TYPE MDP5001_342_I_066CA8C6 :
STRUCT
	MDP5001_342_I1_Channel_Overcurrent						: BIT;
	MDP5001_342_I1_Channel_Inaccurate_Current				: BIT;
	MDP5001_342_I1_Channel_Current_Guard_Warning			: BIT;
	MDP5001_342_I1_Channel_Current_Guard_Error				: BIT;
	MDP5001_342_I1_Channel_Apparent_Power_Guard_Warning		: BIT;
	MDP5001_342_I1_Channel_Apparent_Power_Guard_Error		: BIT;
	MDP5001_342_I1_Channel_Active_Power_Guard_Warning		: BIT;
	MDP5001_342_I1_Channel_Active_Power_Guard_Error			: BIT;
	MDP5001_342_I1_Channel_Reactive_Power_Guard_Warning		: BIT;
	MDP5001_342_I1_Channel_Reactive_Power_Guard_Error		: BIT;
	MDP5001_342_I1_Channel_DPM_Inaccurate					: BIT;
	MDP5001_342_I1_Channel_DPM_Timeout						: BIT;
	MDP5001_342_I1_Channel_TxPDO_Toggle						: BIT;
	MDP5001_342_I1_Channel_Current							: REAL;
	MDP5001_342_I1_Channel_Active_Power						: REAL;
	MDP5001_342_I1_Channel_Apparent_Power					: REAL;
	MDP5001_342_I1_Channel_Reactive_Power_Fundamental		: REAL;
	MDP5001_342_I1_Channel_Active_Energy					: DINT;
	MDP5001_342_I2_Channel_Overcurrent						: BIT;
	MDP5001_342_I2_Channel_Inaccurate_Current				: BIT;
	MDP5001_342_I2_Channel_Current_Guard_Warning			: BIT;
	MDP5001_342_I2_Channel_Current_Guard_Error				: BIT;
	MDP5001_342_I2_Channel_Apparent_Power_Guard_Warning		: BIT;
	MDP5001_342_I2_Channel_Apparent_Power_Guard_Error		: BIT;
	MDP5001_342_I2_Channel_Active_Power_Guard_Warning		: BIT;
	MDP5001_342_I2_Channel_Active_Power_Guard_Error			: BIT;
	MDP5001_342_I2_Channel_Reactive_Power_Guard_Warning		: BIT;
	MDP5001_342_I2_Channel_Reactive_Power_Guard_Error		: BIT;
	MDP5001_342_I2_Channel_DPM_Inaccurate					: BIT;
	MDP5001_342_I2_Channel_DPM_Timeout						: BIT;
	MDP5001_342_I2_Channel_TxPDO_Toggle						: BIT;
	MDP5001_342_I2_Channel_Current							: REAL;
	MDP5001_342_I2_Channel_Active_Power						: REAL;
	MDP5001_342_I2_Channel_Apparent_Power					: REAL;
	MDP5001_342_I2_Channel_Reactive_Power_Fundamental		: REAL;
	MDP5001_342_I2_Channel_Active_Energy					: DINT;
	MDP5001_342_I3_Channel_Overcurrent						: BIT;
	MDP5001_342_I3_Channel_Inaccurate_Current				: BIT;
	MDP5001_342_I3_Channel_Current_Guard_Warning			: BIT;
	MDP5001_342_I3_Channel_Current_Guard_Error				: BIT;
	MDP5001_342_I3_Channel_Apparent_Power_Guard_Warning		: BIT;
	MDP5001_342_I3_Channel_Apparent_Power_Guard_Error		: BIT;
	MDP5001_342_I3_Channel_Active_Power_Guard_Warning		: BIT;
	MDP5001_342_I3_Channel_Active_Power_Guard_Error			: BIT;
	MDP5001_342_I3_Channel_Reactive_Power_Guard_Warning		: BIT;
	MDP5001_342_I3_Channel_Reactive_Power_Guard_Error		: BIT;
	MDP5001_342_I3_Channel_DPM_Inaccurate					: BIT;
	MDP5001_342_I3_Channel_DPM_Timeout						: BIT;
	MDP5001_342_I3_Channel_TxPDO_Toggle						: BIT;
	MDP5001_342_I3_Channel_Current							: REAL;
	MDP5001_342_I3_Channel_Active_Power						: REAL;
	MDP5001_342_I3_Channel_Apparent_Power					: REAL;
	MDP5001_342_I3_Channel_Reactive_Power_Fundamental		: REAL;
	MDP5001_342_I3_Channel_Active_Energy					: DINT;	
	MDP5001_342_I4_Channel_Overcurrent						: BIT;
	MDP5001_342_I4_Channel_Inaccurate_Current				: BIT;
	MDP5001_342_I4_Channel_Current_Guard_Warning			: BIT;
	MDP5001_342_I4_Channel_Current_Guard_Error				: BIT;
	MDP5001_342_I4_Channel_Apparent_Power_Guard_Warning		: BIT;
	MDP5001_342_I4_Channel_Apparent_Power_Guard_Error		: BIT;
	MDP5001_342_I4_Channel_Active_Power_Guard_Warning		: BIT;
	MDP5001_342_I4_Channel_Active_Power_Guard_Error			: BIT;
	MDP5001_342_I4_Channel_Reactive_Power_Guard_Warning		: BIT;
	MDP5001_342_I4_Channel_Reactive_Power_Guard_Error		: BIT;
	MDP5001_342_I4_Channel_DPM_Inaccurate					: BIT;
	MDP5001_342_I4_Channel_DPM_Timeout						: BIT;
	MDP5001_342_I4_Channel_TxPDO_Toggle						: BIT;
	MDP5001_342_I4_Channel_Current							: REAL;
	MDP5001_342_I4_Channel_Active_Power						: REAL;
	MDP5001_342_I4_Channel_Apparent_Power					: REAL;
	MDP5001_342_I4_Channel_Reactive_Power_Fundamental		: REAL;
	MDP5001_342_I4_Channel_Active_Energy					: DINT;	
	MDP5001_342_I5_Channel_Overcurrent						: BIT;
	MDP5001_342_I5_Channel_Inaccurate_Current				: BIT;
	MDP5001_342_I5_Channel_Current_Guard_Warning			: BIT;
	MDP5001_342_I5_Channel_Current_Guard_Error				: BIT;
	MDP5001_342_I5_Channel_Apparent_Power_Guard_Warning		: BIT;
	MDP5001_342_I5_Channel_Apparent_Power_Guard_Error		: BIT;
	MDP5001_342_I5_Channel_Active_Power_Guard_Warning		: BIT;
	MDP5001_342_I5_Channel_Active_Power_Guard_Error			: BIT;
	MDP5001_342_I5_Channel_Reactive_Power_Guard_Warning		: BIT;
	MDP5001_342_I5_Channel_Reactive_Power_Guard_Error		: BIT;
	MDP5001_342_I5_Channel_DPM_Inaccurate					: BIT;
	MDP5001_342_I5_Channel_DPM_Timeout						: BIT;
	MDP5001_342_I5_Channel_TxPDO_Toggle						: BIT;
	MDP5001_342_I5_Channel_Current							: REAL;
	MDP5001_342_I5_Channel_Active_Power						: REAL;
	MDP5001_342_I5_Channel_Apparent_Power					: REAL;
	MDP5001_342_I5_Channel_Reactive_Power_Fundamental		: REAL;
	MDP5001_342_I5_Channel_Active_Energy					: DINT;	
	MDP5001_342_I6_Channel_Overcurrent						: BIT;
	MDP5001_342_I6_Channel_Inaccurate_Current				: BIT;
	MDP5001_342_I6_Channel_Current_Guard_Warning			: BIT;
	MDP5001_342_I6_Channel_Current_Guard_Error				: BIT;
	MDP5001_342_I6_Channel_Apparent_Power_Guard_Warning		: BIT;
	MDP5001_342_I6_Channel_Apparent_Power_Guard_Error		: BIT;
	MDP5001_342_I6_Channel_Active_Power_Guard_Warning		: BIT;
	MDP5001_342_I6_Channel_Active_Power_Guard_Error			: BIT;
	MDP5001_342_I6_Channel_Reactive_Power_Guard_Warning		: BIT;
	MDP5001_342_I6_Channel_Reactive_Power_Guard_Error		: BIT;
	MDP5001_342_I6_Channel_DPM_Inaccurate					: BIT;
	MDP5001_342_I6_Channel_DPM_Timeout						: BIT;
	MDP5001_342_I6_Channel_TxPDO_Toggle						: BIT;
	MDP5001_342_I6_Channel_Current							: REAL;
	MDP5001_342_I6_Channel_Active_Power						: REAL;
	MDP5001_342_I6_Channel_Apparent_Power					: REAL;
	MDP5001_342_I6_Channel_Reactive_Power_Fundamental		: REAL;
	MDP5001_342_I6_Channel_Active_Energy					: DINT;
	MDP5001_342_DPM_Variant_Value_In_TxPDO_Toggle			: BIT;
	MDP5001_342_DPM_Variant_Value_In_Index_1_REAL			: UINT;
	MDP5001_342_DPM_Variant_Value_In_Value_1_REAL			: REAL;
	MDP5001_342_DPM_Variant_Value_In_Index_2_REAL			: UINT; 
	MDP5001_342_DPM_Variant_Value_In_Value_2_REAL			: REAL;
	MDP5001_342_DPM_Variant_Value_In_Index_3_REAL			: UINT;
	MDP5001_342_DPM_Variant_Value_In_Value_3_REAL			: REAL;
	MDP5001_342_DPM_Variant_Value_In_Index_4_ULINT			: UINT;
	MDP5001_342_DPM_Variant_Value_In_Value_4_ULINT			: ULINT;
END_STRUCT
END_TYPE

(* stored: Version 1.1.0.1, ProductVersion 3.1.4024.12
   DUT MDP5001_342_I_066CA8C6: Id {c5cff0ca-927c-4eb3-8c82-f1c6971fead5} *)
